TYPE enum_E:
    (elit_m1, elit_m2);
END_TYPE

(* stored: ProductVersion 3.1.0.18, Version 1.1.0.1 *)
